(* IEC 61131-3 sources: RL_MAR/experiments/comparison/llm4plc/results/deepseek-ai-DeepSeek-V3.2_20260506_104945/20260506_115646, 4 files *)

(* ---- generated_code_iteration_0.st ---- *)
START_ST
FUNCTION_BLOCK WindowCleaningSystem
VAR_INPUT
    StartButton : BOOL;
    EmergencyStop : BOOL;
    UpperLimit : BOOL;
    LowerLimit : BOOL;
END_VAR

VAR_OUTPUT
    ElevatorUp : BOOL;
    ElevatorDown : BOOL;
    RotateClockwise : BOOL;
    WaterPump : BOOL;
END_VAR

VAR
    CleaningInProgress : BOOL;
    state : INT;
    prevState : INT;
END_VAR

(* State definitions *)
CONST
    STATE_IDLE : INT := 0;
    STATE_MOVING_UP : INT := 1;
    STATE_CLEANING_DOWN : INT := 2;
    STATE_EMERGENCY_STOP : INT := 3;
END_CONST

(* Main FSM execution *)
IF EmergencyStop = TRUE THEN
    state := STATE_EMERGENCY_STOP;
ELSE
    CASE state OF
        STATE_IDLE:
            IF StartButton = TRUE AND NOT CleaningInProgress THEN
                state := STATE_MOVING_UP;
            END_IF;

        STATE_MOVING_UP:
            IF UpperLimit = TRUE THEN
                state := STATE_CLEANING_DOWN;
            END_IF;

        STATE_CLEANING_DOWN:
            IF LowerLimit = TRUE THEN
                state := STATE_IDLE;
            END_IF;

        STATE_EMERGENCY_STOP:
            (* Remain in emergency stop until EmergencyStop is released *)
            IF EmergencyStop = FALSE THEN
                state := STATE_IDLE;
            END_IF;
    END_CASE;
END_IF;

(* Manage CleaningInProgress flag *)
IF state = STATE_MOVING_UP AND prevState = STATE_IDLE THEN
    CleaningInProgress := TRUE;
ELSIF (state = STATE_IDLE AND prevState = STATE_CLEANING_DOWN) OR
      (state = STATE_EMERGENCY_STOP AND prevState <> STATE_EMERGENCY_STOP) THEN
    CleaningInProgress := FALSE;
END_IF;

(* Set outputs based on current state *)
CASE state OF
    STATE_IDLE:
        ElevatorUp := FALSE;
        ElevatorDown := FALSE;
        RotateClockwise := FALSE;
        WaterPump := FALSE;

    STATE_MOVING_UP:
        ElevatorUp := TRUE;
        ElevatorDown := FALSE;
        RotateClockwise := FALSE;
        WaterPump := FALSE;

    STATE_CLEANING_DOWN:
        ElevatorUp := FALSE;
        ElevatorDown := TRUE;
        RotateClockwise := TRUE;
        WaterPump := TRUE;

    STATE_EMERGENCY_STOP:
        ElevatorUp := FALSE;
        ElevatorDown := FALSE;
        RotateClockwise := FALSE;
        WaterPump := FALSE;
END_CASE;

(* Store previous state for edge detection *)
prevState := state;

END_FUNCTION_BLOCK
END_ST

(* ---- generated_code_iteration_1.st ---- *)
START_REASON
The feedback indicates a syntax error in the CODESYS compiler validation: "应该用';' 替换'STATE_IDLE'". This is Chinese for "should replace 'STATE_IDLE' with ';'". This suggests that in the CONST section, the constant definition for STATE_IDLE is incorrectly terminated. In Structured Text, constant definitions should end with a semicolon (;), not a colon or other punctuation. Looking at the original code:

CONST
    STATE_IDLE : INT := 0;
    STATE_MOVING_UP : INT := 1;
    STATE_CLEANING_DOWN : INT := 2;
    STATE_EMERGENCY_STOP : INT := 3;
END_CONST

All lines appear to end with semicolons, but the feedback specifically points to STATE_IDLE. Possibly, there's a hidden character or formatting issue in the original submission that caused the compiler to misinterpret the line. To fix this, I'll ensure that the CONST section is correctly formatted with proper semicolons and no extraneous characters. I'll rewrite the CONST section clearly, ensuring each constant definition ends with a semicolon. Additionally, I'll verify the overall structure to prevent any other potential syntax issues.

The rest of the code structure seems correct: it uses FUNCTION_BLOCK, proper variable sections with END_VAR, and a state machine. No changes are needed to the logic, but I'll ensure the code is clean and adheres to ST standards.
END_REASON

START_ST
FUNCTION_BLOCK WindowCleaningSystem
VAR_INPUT
    StartButton : BOOL;
    EmergencyStop : BOOL;
    UpperLimit : BOOL;
    LowerLimit : BOOL;
END_VAR

VAR_OUTPUT
    ElevatorUp : BOOL;
    ElevatorDown : BOOL;
    RotateClockwise : BOOL;
    WaterPump : BOOL;
END_VAR

VAR
    CleaningInProgress : BOOL;
    state : INT;
    prevState : INT;
END_VAR

(* State definitions *)
CONST
    STATE_IDLE : INT := 0;
    STATE_MOVING_UP : INT := 1;
    STATE_CLEANING_DOWN : INT := 2;
    STATE_EMERGENCY_STOP : INT := 3;
END_CONST

(* Main FSM execution *)
IF EmergencyStop = TRUE THEN
    state := STATE_EMERGENCY_STOP;
ELSE
    CASE state OF
        STATE_IDLE:
            IF StartButton = TRUE AND NOT CleaningInProgress THEN
                state := STATE_MOVING_UP;
            END_IF;

        STATE_MOVING_UP:
            IF UpperLimit = TRUE THEN
                state := STATE_CLEANING_DOWN;
            END_IF;

        STATE_CLEANING_DOWN:
            IF LowerLimit = TRUE THEN
                state := STATE_IDLE;
            END_IF;

        STATE_EMERGENCY_STOP:
            (* Remain in emergency stop until EmergencyStop is released *)
            IF EmergencyStop = FALSE THEN
                state := STATE_IDLE;
            END_IF;
    END_CASE;
END_IF;

(* Manage CleaningInProgress flag *)
IF state = STATE_MOVING_UP AND prevState = STATE_IDLE THEN
    CleaningInProgress := TRUE;
ELSIF (state = STATE_IDLE AND prevState = STATE_CLEANING_DOWN) OR
      (state = STATE_EMERGENCY_STOP AND prevState <> STATE_EMERGENCY_STOP) THEN
    CleaningInProgress := FALSE;
END_IF;

(* Set outputs based on current state *)
CASE state OF
    STATE_IDLE:
        ElevatorUp := FALSE;
        ElevatorDown := FALSE;
        RotateClockwise := FALSE;
        WaterPump := FALSE;

    STATE_MOVING_UP:
        ElevatorUp := TRUE;
        ElevatorDown := FALSE;
        RotateClockwise := FALSE;
        WaterPump := FALSE;

    STATE_CLEANING_DOWN:
        ElevatorUp := FALSE;
        ElevatorDown := TRUE;
        RotateClockwise := TRUE;
        WaterPump := TRUE;

    STATE_EMERGENCY_STOP:
        ElevatorUp := FALSE;
        ElevatorDown := FALSE;
        RotateClockwise := FALSE;
        WaterPump := FALSE;
END_CASE;

(* Store previous state for edge detection *)
prevState := state;

END_FUNCTION_BLOCK
END_ST

(* ---- generated_code_iteration_2.st ---- *)
START_REASON
The feedback indicates an encoding issue with the CODESYS compiler validation: "gbk' codec can't decode byte 0xaf in position 93: illegal multibyte sequence". This suggests that there are non-ASCII characters or special characters in the code that the compiler cannot decode properly. The error occurs at position 93, which likely points to a specific character in the code. Given the previous code, the issue might be in the comment sections or variable names that contain non-standard characters. Since the code is in English, the problem could be with the comment delimiters or hidden characters introduced during copying. To fix this, I will ensure all comments use standard ASCII characters and remove any potential non-ASCII characters. I'll rewrite the code with clean comments and verify that all text is within the ASCII range. Additionally, I'll ensure the structure is correct to prevent any syntax errors.
END_REASON

START_ST
FUNCTION_BLOCK WindowCleaningSystem
VAR_INPUT
    StartButton : BOOL;
    EmergencyStop : BOOL;
    UpperLimit : BOOL;
    LowerLimit : BOOL;
END_VAR

VAR_OUTPUT
    ElevatorUp : BOOL;
    ElevatorDown : BOOL;
    RotateClockwise : BOOL;
    WaterPump : BOOL;
END_VAR

VAR
    CleaningInProgress : BOOL;
    state : INT;
    prevState : INT;
END_VAR

CONST
    STATE_IDLE : INT := 0;
    STATE_MOVING_UP : INT := 1;
    STATE_CLEANING_DOWN : INT := 2;
    STATE_EMERGENCY_STOP : INT := 3;
END_CONST

IF EmergencyStop = TRUE THEN
    state := STATE_EMERGENCY_STOP;
ELSE
    CASE state OF
        STATE_IDLE:
            IF StartButton = TRUE AND NOT CleaningInProgress THEN
                state := STATE_MOVING_UP;
            END_IF;

        STATE_MOVING_UP:
            IF UpperLimit = TRUE THEN
                state := STATE_CLEANING_DOWN;
            END_IF;

        STATE_CLEANING_DOWN:
            IF LowerLimit = TRUE THEN
                state := STATE_IDLE;
            END_IF;

        STATE_EMERGENCY_STOP:
            IF EmergencyStop = FALSE THEN
                state := STATE_IDLE;
            END_IF;
    END_CASE;
END_IF;

IF state = STATE_MOVING_UP AND prevState = STATE_IDLE THEN
    CleaningInProgress := TRUE;
ELSIF (state = STATE_IDLE AND prevState = STATE_CLEANING_DOWN) OR
      (state = STATE_EMERGENCY_STOP AND prevState <> STATE_EMERGENCY_STOP) THEN
    CleaningInProgress := FALSE;
END_IF;

CASE state OF
    STATE_IDLE:
        ElevatorUp := FALSE;
        ElevatorDown := FALSE;
        RotateClockwise := FALSE;
        WaterPump := FALSE;

    STATE_MOVING_UP:
        ElevatorUp := TRUE;
        ElevatorDown := FALSE;
        RotateClockwise := FALSE;
        WaterPump := FALSE;

    STATE_CLEANING_DOWN:
        ElevatorUp := FALSE;
        ElevatorDown := TRUE;
        RotateClockwise := TRUE;
        WaterPump := TRUE;

    STATE_EMERGENCY_STOP:
        ElevatorUp := FALSE;
        ElevatorDown := FALSE;
        RotateClockwise := FALSE;
        WaterPump := FALSE;
END_CASE;

prevState := state;

END_FUNCTION_BLOCK
END_ST

(* ---- generated_code_iteration_3.st ---- *)
START_REASON
The feedback indicates a CODESYS compiler validation error: "应该用';' 替换'STATE_IDLE'", which translates to "should replace 'STATE_IDLE' with ';'". This suggests a syntax issue in the CONST declaration section. In CODESYS Structured Text, CONST declarations should end with semicolons (;) after each constant assignment, not colons (:). Looking at the previous code, I wrote "STATE_IDLE : INT := 0;" but the feedback points to 'STATE_IDLE' specifically, implying the colon after STATE_IDLE might be incorrect. However, the standard syntax for CONST is "CONSTANT_NAME : DATA_TYPE := VALUE;". The error might be due to a misinterpretation or a specific CODESYS version requirement. To fix this, I'll ensure all CONST declarations use proper syntax with semicolons and verify the structure. I'll also check for any missing semicolons or incorrect punctuation in the CONST section.
END_REASON

START_ST
FUNCTION_BLOCK WindowCleaningSystem
VAR_INPUT
    StartButton : BOOL;
    EmergencyStop : BOOL;
    UpperLimit : BOOL;
    LowerLimit : BOOL;
END_VAR

VAR_OUTPUT
    ElevatorUp : BOOL;
    ElevatorDown : BOOL;
    RotateClockwise : BOOL;
    WaterPump : BOOL;
END_VAR

VAR
    CleaningInProgress : BOOL;
    state : INT;
    prevState : INT;
END_VAR

CONST
    STATE_IDLE : INT := 0;
    STATE_MOVING_UP : INT := 1;
    STATE_CLEANING_DOWN : INT := 2;
    STATE_EMERGENCY_STOP : INT := 3;
END_CONST

IF EmergencyStop = TRUE THEN
    state := STATE_EMERGENCY_STOP;
ELSE
    CASE state OF
        STATE_IDLE:
            IF StartButton = TRUE AND NOT CleaningInProgress THEN
                state := STATE_MOVING_UP;
            END_IF;

        STATE_MOVING_UP:
            IF UpperLimit = TRUE THEN
                state := STATE_CLEANING_DOWN;
            END_IF;

        STATE_CLEANING_DOWN:
            IF LowerLimit = TRUE THEN
                state := STATE_IDLE;
            END_IF;

        STATE_EMERGENCY_STOP:
            IF EmergencyStop = FALSE THEN
                state := STATE_IDLE;
            END_IF;
    END_CASE;
END_IF;

IF state = STATE_MOVING_UP AND prevState = STATE_IDLE THEN
    CleaningInProgress := TRUE;
ELSIF (state = STATE_IDLE AND prevState = STATE_CLEANING_DOWN) OR
      (state = STATE_EMERGENCY_STOP AND prevState <> STATE_EMERGENCY_STOP) THEN
    CleaningInProgress := FALSE;
END_IF;

CASE state OF
    STATE_IDLE:
        ElevatorUp := FALSE;
        ElevatorDown := FALSE;
        RotateClockwise := FALSE;
        WaterPump := FALSE;

    STATE_MOVING_UP:
        ElevatorUp := TRUE;
        ElevatorDown := FALSE;
        RotateClockwise := FALSE;
        WaterPump := FALSE;

    STATE_CLEANING_DOWN:
        ElevatorUp := FALSE;
        ElevatorDown := TRUE;
        RotateClockwise := TRUE;
        WaterPump := TRUE;

    STATE_EMERGENCY_STOP:
        ElevatorUp := FALSE;
        ElevatorDown := FALSE;
        RotateClockwise := FALSE;
        WaterPump := FALSE;
END_CASE;

prevState := state;

END_FUNCTION_BLOCK
END_ST
